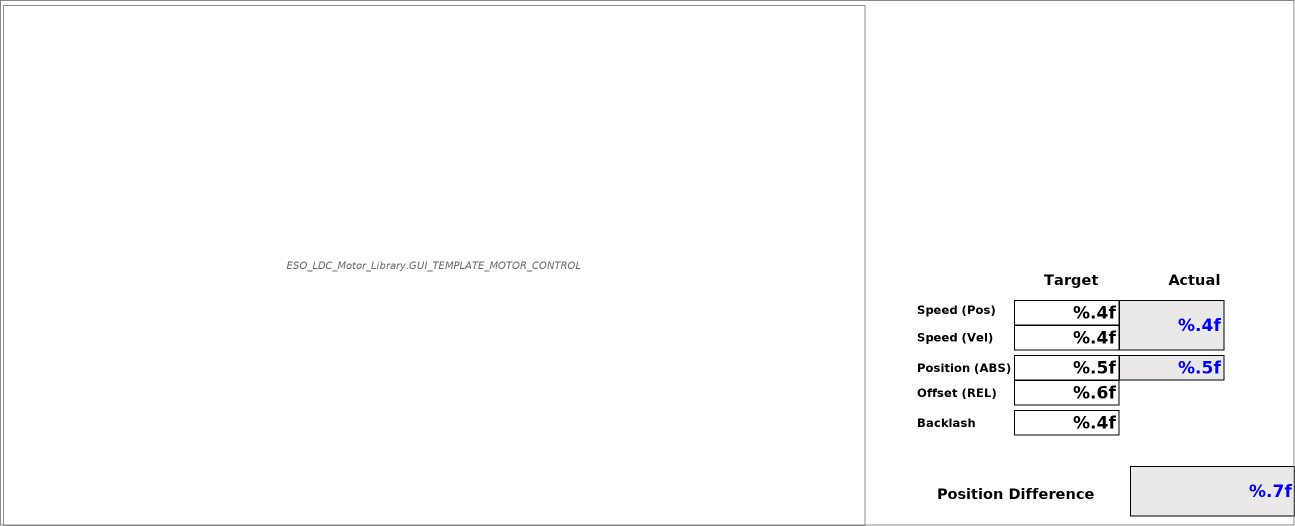
VISUALIZATION DL_Servo_1_Control  // 1295x526
    Frame (3,5 862x521)
        shows ESO_LDC_Motor_Library.GUI_TEMPLATE_MOTOR_CONTROL(m_Instance := MAIN.DL_Servo_1)
    Rectangle (914,300 95x20), "Speed (Pos)"
    Rectangle (1119,355 105x25), "%.5f", text variable: MAIN.DL_Servo_1.stat.lrPosActual, input disabled if: false
    Rectangle (1041,270 190x20), "Target Actual"
    Rectangle (914,358 95x20), "Position (ABS)"
    Rectangle (1119,300 105x50), "%.4f", text variable: MAIN.DL_Servo_1.stat.lrVelActual, input disabled if: false
    Rectangle (1014,325 105x25), "%.4f", text variable: MAIN.DL_Servo_1.ctrl.lrVelocity
        OnMouseDown: write the text variable via Default
    Rectangle (914,413 95x20), "Backlash"
    Rectangle (1014,410 105x25), "%.4f", text variable: MAIN.DL_Servo_1.cfg.lrBacklash
        OnMouseDown: write the text variable via Default
    Rectangle (914,325 95x25), "Speed (Vel)"
    Rectangle (1014,355 105x25), "%.5f", tooltip "Absolute position used by "MOVE ABS"", text variable: MAIN.DL_Servo_1.ctrl.lrPosition
        OnMouseDown: write the text variable via Default
    Rectangle (1014,300 105x25), "%.4f", text variable: MAIN.DL_Servo_1.cfg.lrDefaultVelocity
        OnMouseDown: write the text variable via Default
    Rectangle (914,383 95x20), "Offset (REL)"
    Rectangle (1014,380 105x25), "%.6f", tooltip "Relative offset used by "MOVE REL"", text variable: MAIN.DL_Servo_1.ctrl.lrOffset
        OnMouseDown: write the text variable via Default
    Rectangle (1130,466 165x50), "%.7f", text variable: MAIN.DL_Servo_1.stat.lrPosError, input disabled if: false
    Rectangle (934,484 190x20), "Position Difference"
END_VISUALIZATION

(* stored: Version 1.1.0.1, ProductVersion 3.1.4024.12
   Visu DL_Servo_1_Control: Id {2936fa0d-e441-4b95-844b-d6b3facffedb} *)
